SUBAPPLICATION Uebung_020i_AX (* DigitalInput_I1 auf DigitalOutput_Q1; AX_PULSE; Teach-In *)
  (* Standard: 61499-2; Description: Copyright (c) 2023 Meisterschulen am Ostbahnhof This program and the accompanying materials are made available under the terms of the Eclipse Public License 2.0 which is available at https://www.eclipse.org/legal/epl-2.0/ SPDX-License-Identifier: EPL-2.0 *)
  (* Version 1.0, 2026-01-16, Franz Höpfinger, Meisterschulen am Ostbahnhof, initial API and implementation and/or initial documentation *)
  PACKAGE Uebungen;
  IMPORT logiBUS::io::DI::logiBUS_DI::Input_I1;
  IMPORT logiBUS::io::DI::logiBUS_DI::Input_I2;
  IMPORT logiBUS::io::DI::logiBUS_DI_Events::BUTTON_SINGLE_CLICK;
  IMPORT logiBUS::io::DQ::logiBUS_DO::Output_Q1;
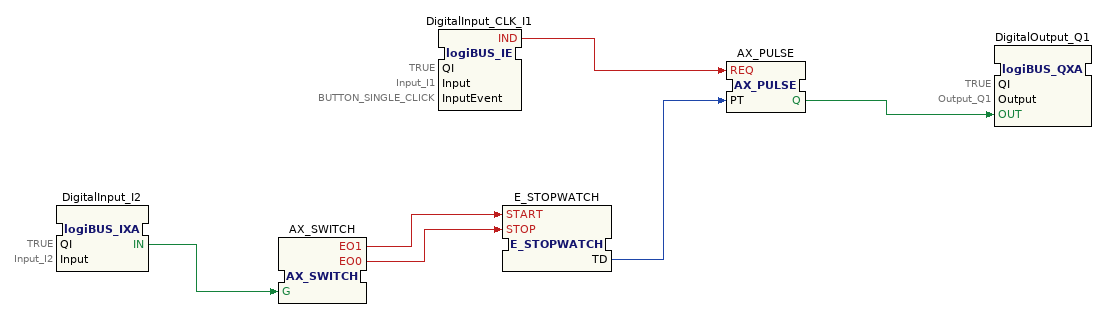
  FBS
    DigitalInput_CLK_I1 : logiBUS::io::DI::logiBUS_IE(QI := TRUE, Input := Input_I1, InputEvent := BUTTON_SINGLE_CLICK);
    AX_PULSE : adapter::events::unidirectional::timers::AX_PULSE;
    DigitalOutput_Q1 : logiBUS::io::DQ::logiBUS_QXA(QI := TRUE, Output := Output_Q1);
    DigitalInput_I2 : logiBUS::io::DI::logiBUS_IXA(QI := TRUE, Input := Input_I2);
    AX_SWITCH : adapter::events::unidirectional::AX_SWITCH;
    E_STOPWATCH : eclipse4diac::utils::timing::E_STOPWATCH;
  END_FBS
  EVENT_CONNECTIONS
    DigitalInput_CLK_I1.IND TO AX_PULSE.REQ;
    AX_SWITCH.EO1 TO E_STOPWATCH.START;
    AX_SWITCH.EO0 TO E_STOPWATCH.STOP;
  END_CONNECTIONS
  DATA_CONNECTIONS
    E_STOPWATCH.TD TO AX_PULSE.PT;
  END_CONNECTIONS
  ADAPTER_CONNECTIONS
    AX_PULSE.Q TO DigitalOutput_Q1.OUT;
    DigitalInput_I2.IN TO AX_SWITCH.G;
  END_CONNECTIONS
END_SUBAPPLICATION
